{attribute addProperty BoxType "EPP5101-0011-0016"}
{attribute addProperty Id "StatusAT %I*Status_1B2A8E891621Counter_valueAT %I*UINT16217Latch_valueAT %I*UINT16218"}
{attribute addProperty CRC "1026846327"}
{attribute addProperty SizeInBites "48"}
{attribute addProperty SizeInBytes "6"}
TYPE ENC_Status_compact_3D346E77 :
STRUCT
	{attribute addProperty Name "Status"}
	Status AT %I* : Status_1B2A8E89;
	{attribute addProperty Name "Counter_value"}
	Counter_value AT %I* : UINT;
	{attribute addProperty Name "Latch_value"}
	Latch_value AT %I* : UINT;
END_STRUCT
END_TYPE

(* stored: Version 1.2.0.0, ProductVersion 3.1.4024.9
   DUT ENC_Status_compact_3D346E77: Id {26f218b7-c2eb-4f98-a95e-c28bbe6d04c2} *)
